// TIA Portal V20 export
TYPE "typeScrapBoxCommands"
// stored: Access Published, IsFailsafeCompliant true, Namespace Safety
   STRUCT
      lock : Bool;
      unlock : Bool;
      reset : Bool;
   END_STRUCT;
END_TYPE
